FUNCTION_BLOCK FB_Syntax_Action
VAR
    _nCounter : INT;
END_VAR

_nCounter := _nCounter + 1;

ACTION A_Reset:
_nCounter := 0;
END_ACTION

END_FUNCTION_BLOCK

(* stored: Version 1.1.0.1, ProductVersion 3.1.4024.16
   POU FB_Syntax_Action: Id {0efbec70-18ed-41e5-a179-e4fee62f3278}, SpecialFunc None
   Action A_Reset: Id {151a03be-b987-4adc-ae5a-9f21f38aeda5} *)
